FUNCTION_BLOCK FB_VALVE_X_3_PROP IMPLEMENTS I_VALVE_X_3_PROP
VAR_OUTPUT
  iAnalogSwitch:                                          INT;
END_VAR
VAR //General
	{attribute 'instance-path'} 
  {attribute 'noinit'} 
	strInstancePath:									                      STRING;
	bInit: 												                          BOOL:=TRUE;
	strFullObjectPath: 								                      STRING;
	stEvent:											                          ST_EVENT;
	bAck:												                            BOOL;
END_VAR
VAR   // From FB_init	
	itfLogEvents: 										                      I_HANDLE_EVENTS;
  itfOpMode:											                        I_OP_MODE;
END_VAR                                      				
VAR	// Step chain control                				
  eSeq, eLastSeq, eNextSeq:					                      E_SEQ_VALVE; 
                  				
  //eActiveSeqState, eLastActiveSeqState:                 E_SEQ_GENERAL;
	(*
  iInternalSeqStateCase, iLastInternalSeqStateCase:       INT:=0;       
	tonDelay, tonTimeOut, tonStepTime:						          TON;
	tDelay:													                        TIME := T#100MS;
	tTimeOut:												                        TIME := T#100MS;
	tTimeOutExt:											                      TIME := T#100MS;
	bDelayActive, bTimeOutActiveQuit, bTimeOutActiveNoQuit:	BOOL;//Timer Option
	bActiveStep, bDebugAcitve, bDebugNext:					        BOOL;//Debug Option
	i:														                          INT;
 	iError:													                        INT; //ERROR-CODE                    	                   		
	listLastSteps:											                    ARRAY[0..49] OF ST_LAST_STEPS;	
	strExtraInfo:											                      STRING; 
	eStep_Type:												                      E_STEP_STATE_TYPE; 
	bDebugModeActive:										                    BOOL;   
	bWaitForBreakpoint:										                  BOOL;
	bBreakpointActive:										                  BOOL;
	bDebugResume:											                      BOOL;   
	listBreakpoint:											                    ARRAY[0..10] OF  INT;    
*)
i:														                            INT;
stSeqCtrlGeneral:											                    ST_SEQ_CTRL_GEN;     	
END_VAR                                             		
VAR                                                 		
	bMethodeFromExtStarted:									                BOOL;
	bMethodeFromExtActive:									                BOOL;
	bMethodeFromExtDone:									                  BOOL;
	strTemp:												                        STRING;
END_VAR   
VAR
  stHMI:                                                  ST_HMI_VALVE;
  tDelay:                                                 TIME;
  rSpeedInPercent:                                        REAL;
END_VAR
VAR
  iOutputVal:                                             INT; 
END_VAR                 	
VAR_TEMP                    	
	iTemp:										                              INT;
END_VAR

// Set FBs and Interfaces ready after switch internal step
IF stSeqCtrlGeneral.iInternalSeqStateCase <> stSeqCtrlGeneral.iLastInternalSeqStateCase AND NOT stSeqCtrlGeneral.bExitSetReadyState THEN
  IF TRUE
  //AND ...
  THEN
    stSeqCtrlGeneral.bExitSetReadyState := TRUE;
  ELSE
    RETURN;
  END_IF
END_IF

stSeqCtrlGeneral.strObject := F_CreateObjectName(strInstancePath);

// First method call
_m_SequenceManager();
//_m_SaveLastStep();

CASE eSeq OF 
  E_SEQ_VALVE.BASE:;
  
	E_SEQ_VALVE.INIT: _m_Seq_INIT();
		IF TRUE
		AND (stSeqCtrlGeneral.eActiveSeqState = E_SEQ_GENERAL.DONE) 
		THEN
			eSeq := E_SEQ_VALVE.BASE;
		END_IF
		
	E_SEQ_VALVE.SETUP:;
  
	// Process
  E_SEQ_VALVE.SET_LIMIT: _m_Seq_VALVE_CTRL();
    IF TRUE
		AND (stSeqCtrlGeneral.eActiveSeqState = E_SEQ_GENERAL.DONE) 
		THEN
			eSeq := E_SEQ_VALVE.BASE;
		END_IF
    
  E_SEQ_VALVE.SET_LIMIT_SMOOTH: _m_Seq_VALVE_CTRL_SMOOTH();
    IF TRUE
		AND (stSeqCtrlGeneral.eActiveSeqState = E_SEQ_GENERAL.DONE) 
		THEN
			eSeq := E_SEQ_VALVE.BASE;
		END_IF

  // End
	E_SEQ_VALVE.END:;
	E_SEQ_VALVE.ERROR_SEQ:;	
END_CASE

strTemp:=TO_STRING(eSeq);

METHOD PRIVATE _m_DebugManager
VAR_INPUT
	iStepID: int;
END_VAR
IF TRUE
AND THIS^.stSeqCtrlGeneral.bDebugModeActive 
AND NOT THIS^.stSeqCtrlGeneral.bActiveStep
THEN


THIS^.stSeqCtrlGeneral.bBreakpointActive:=FALSE;

FOR i:=0 TO 10 DO
	
	IF TRUE
	AND iStepID=THIS^.stSeqCtrlGeneral.listBreakpoint[i] 
	AND iStepID<>0
	THEN
		EXIT;
	END_IF
END_FOR
IF (i<=10) THEN
	THIS^.stSeqCtrlGeneral.bBreakpointActive:=TRUE;
END_IF

END_IF
END_METHOD

METHOD PRIVATE _m_Delay : BOOL
VAR_INPUT
	DelayTime:	TIME;
END_VAR
THIS^.stSeqCtrlGeneral.bDelayActive:=TRUE;
THIS^.stSeqCtrlGeneral.tDelay:=DelayTime;
_m_Delay:=FALSE;
IF THIS^.stSeqCtrlGeneral.tonDelay.Q THEN
	_m_Delay:=TRUE;
END_IF
END_METHOD

METHOD PRIVATE _m_GeneralStepSetting : BOOL
VAR_INPUT
	StepType:			    	E_STEP_STATE_TYPE;
	InfoTextID:					STRING(20);
	EnableDebug:	   			BOOL;	
	
END_VAR
IF THIS^.stSeqCtrlGeneral.bActiveStep THEN
	THIS^.stSeqCtrlGeneral.eStep_Type:=StepType;
	THIS^.stSeqCtrlGeneral.strExtraInfo:= GenLib.F_RET_TXTLIST_ENTRY(strPortNr:='851',strID:='',strTxtLstName:=InfoTextID);
END_IF
END_METHOD

METHOD PRIVATE _m_SaveLastStep : BOOL
VAR_INPUT
END_VAR
VAR
	i: dint;
END_VAR
IF NOT THIS^.stSeqCtrlGeneral.bActiveStep THEN
	
	FOR i:=49 TO 1 BY -1 DO
			stSeqCtrlGeneral.listLastSteps[i].strStepName:=stSeqCtrlGeneral.listLastSteps[i-1].strStepName;
			stSeqCtrlGeneral.listLastSteps[i].tStepTime:=stSeqCtrlGeneral.listLastSteps[i-1].tStepTime;
			stSeqCtrlGeneral.listLastSteps[i].tDelayTime:=stSeqCtrlGeneral.listLastSteps[i-1].tDelayTime;
	END_FOR
	stSeqCtrlGeneral.listLastSteps[0].strStepName:=TO_STRING(THIS^.eSeq);
	stSeqCtrlGeneral.listLastSteps[1].tStepTime:=THIS^.stSeqCtrlGeneral.tonStepTime.ET;
	stSeqCtrlGeneral.listLastSteps[1].tStepTime:=THIS^.stSeqCtrlGeneral.tonDelay.ET;
ELSE
	stSeqCtrlGeneral.listLastSteps[0].tStepTime:=THIS^.stSeqCtrlGeneral.tonStepTime.ET;
	stSeqCtrlGeneral.listLastSteps[0].tDelayTime:=THIS^.stSeqCtrlGeneral.tonDelay.ET;	
END_IF
END_METHOD

METHOD PRIVATE _m_Seq_INIT : BOOL
VAR
  ActiveSeq: STRING;
END_VAR
//THIS^._m_GeneralStepSetting(StepType:=E_STEP_STATE_TYPE.INIT,
ActiveSeq := TO_STRING(THIS^.eSeq);

CASE THIS^.stSeqCtrlGeneral.eActiveSeqState OF
E_SEQ_GENERAL.READY:;

	
E_SEQ_GENERAL.EXECUTE:;
	IF TRUE
	THEN
		THIS^.stSeqCtrlGeneral.eActiveSeqState := E_SEQ_GENERAL.RESET;
	END_IF
  
E_SEQ_GENERAL.RESET:;
	stSeqCtrlGeneral.iInternalSeqStateCase := 0;
	IF TRUE
	THEN
		THIS^.stSeqCtrlGeneral.eActiveSeqState := E_SEQ_GENERAL.BUSY;
	END_IF
  
E_SEQ_GENERAL.BUSY:;
	CASE THIS^.stSeqCtrlGeneral.iInternalSeqStateCase OF
    0:  // Reset valve
      IF TRUE 
			THEN 
        iAnalogSwitch := 0;
        IF _m_Delay(T#1S) THEN
          THIS^.stSeqCtrlGeneral.iInternalSeqStateCase := 1000;
				END_IF
			END_IF
      
	ELSE
		THIS^.stSeqCtrlGeneral.eActiveSeqState := E_SEQ_GENERAL.DONE;  
	END_CASE
	THIS^.stSeqCtrlGeneral.strExtraInfo := CONCAT('Internal state: ', TO_STRING(THIS^.stSeqCtrlGeneral.iInternalSeqStateCase));

E_SEQ_GENERAL.DONE:;

E_SEQ_GENERAL.ERROR:;

E_SEQ_GENERAL.TIME_OUT:; 
IF TRUE
AND THIS^.stSeqCtrlGeneral.bTimeOutActiveQuit 
THEN
  THIS^.stSeqCtrlGeneral.strExtraInfo := 'Bitte quittieren und erneut testen';
  IF TRUE
  //AND itfOpMode.P_QUIT
  THEN
    THIS^.stSeqCtrlGeneral.eActiveSeqState := E_SEQ_GENERAL.EXECUTE;
	END_IF
  
END_IF

ELSE
  THIS^.stSeqCtrlGeneral.eActiveSeqState := E_SEQ_GENERAL.ERROR;
END_CASE
END_METHOD

METHOD PRIVATE _m_Seq_VALVE_CTRL : BOOL
VAR
  ActiveSeq:  STRING;
END_VAR
//THIS^._m_GeneralStepSetting(StepType:=E_STEP_STATE_TYPE.INIT,
ActiveSeq := TO_STRING(THIS^.eSeq);

CASE THIS^.stSeqCtrlGeneral.eActiveSeqState OF
E_SEQ_GENERAL.READY:;

	
E_SEQ_GENERAL.EXECUTE:;
	IF TRUE
	THEN
		THIS^.stSeqCtrlGeneral.eActiveSeqState := E_SEQ_GENERAL.RESET;
	END_IF
  
E_SEQ_GENERAL.RESET:;
	stSeqCtrlGeneral.iInternalSeqStateCase := 0;
	IF TRUE
	THEN
		THIS^.stSeqCtrlGeneral.eActiveSeqState := E_SEQ_GENERAL.BUSY;
	END_IF
  
E_SEQ_GENERAL.BUSY:;
	CASE THIS^.stSeqCtrlGeneral.iInternalSeqStateCase OF
    0:  // Calc output value
      IF TRUE 
			THEN 
        THIS^.iOutputVal := TO_INT(327.67 * THIS^.rSpeedInPercent);
        IF THIS^.iOutputVal < 0 THEN 
          THIS^.iOutputVal := THIS^.iOutputVal - 1;
        END_IF
        iAnalogSwitch := THIS^.iOutputVal;
        THIS^.stSeqCtrlGeneral.iInternalSeqStateCase := 10;
			END_IF
      
    10:  // Set output value
      IF TRUE 
			THEN 
        iAnalogSwitch := THIS^.iOutputVal;
        THIS^.stSeqCtrlGeneral.iInternalSeqStateCase := 1000;
			END_IF
      
	ELSE
		THIS^.stSeqCtrlGeneral.eActiveSeqState := E_SEQ_GENERAL.DONE;  
	END_CASE
	THIS^.stSeqCtrlGeneral.strExtraInfo := CONCAT('Internal state: ', TO_STRING(THIS^.stSeqCtrlGeneral.iInternalSeqStateCase));

E_SEQ_GENERAL.DONE:;

E_SEQ_GENERAL.ERROR:;

E_SEQ_GENERAL.TIME_OUT:; 
IF TRUE
AND THIS^.stSeqCtrlGeneral.bTimeOutActiveQuit 
THEN
  THIS^.stSeqCtrlGeneral.strExtraInfo := 'Bitte quittieren und erneut testen';
  IF TRUE
  //AND itfOpMode.P_QUIT
  THEN
    THIS^.stSeqCtrlGeneral.eActiveSeqState := E_SEQ_GENERAL.EXECUTE;
	END_IF
  
END_IF

ELSE
  THIS^.stSeqCtrlGeneral.eActiveSeqState := E_SEQ_GENERAL.ERROR;
END_CASE
END_METHOD

METHOD PRIVATE _m_Seq_VALVE_CTRL_SMOOTH : BOOL
VAR
  ActiveSeq:  STRING;
END_VAR
//THIS^._m_GeneralStepSetting(StepType:=E_STEP_STATE_TYPE.INIT,
ActiveSeq := TO_STRING(THIS^.eSeq);

CASE THIS^.stSeqCtrlGeneral.eActiveSeqState OF
E_SEQ_GENERAL.READY:;

	
E_SEQ_GENERAL.EXECUTE:;
	IF TRUE
	THEN
		THIS^.stSeqCtrlGeneral.eActiveSeqState := E_SEQ_GENERAL.RESET;
	END_IF
  
E_SEQ_GENERAL.RESET:;
	stSeqCtrlGeneral.iInternalSeqStateCase := 0;
	IF TRUE
	THEN
		THIS^.stSeqCtrlGeneral.eActiveSeqState := E_SEQ_GENERAL.BUSY;
	END_IF
  
E_SEQ_GENERAL.BUSY:;
	CASE THIS^.stSeqCtrlGeneral.iInternalSeqStateCase OF
    0:  // Calc output value
      IF TRUE 
			THEN 
        THIS^.iOutputVal := TO_INT(327.67 * THIS^.rSpeedInPercent);
        IF THIS^.iOutputVal < 0 THEN 
          THIS^.iOutputVal := THIS^.iOutputVal - 1;
        END_IF
        iAnalogSwitch := THIS^.iOutputVal;
        THIS^.stSeqCtrlGeneral.iInternalSeqStateCase := 10;
			END_IF
      
    10:  // Set output value
      IF TRUE 
			THEN 
        IF iAnalogSwitch > THIS^.iOutputVal + 100 THEN
          iAnalogSwitch := iAnalogSwitch - 100;
        ELSIF iAnalogSwitch < THIS^.iOutputVal - 100 THEN
          iAnalogSwitch := iAnalogSwitch + 100;
        END_IF
        IF ABS(iAnalogSwitch - THIS^.iOutputVal) <= 100 THEN
          THIS^.stSeqCtrlGeneral.iInternalSeqStateCase := 20;
        END_IF
			END_IF
      
    20:  // Set output value
      IF TRUE 
			THEN 
        iAnalogSwitch := THIS^.iOutputVal;
        THIS^.stSeqCtrlGeneral.iInternalSeqStateCase := 1000;
			END_IF
      
	ELSE
		THIS^.stSeqCtrlGeneral.eActiveSeqState := E_SEQ_GENERAL.DONE;  
	END_CASE
	THIS^.stSeqCtrlGeneral.strExtraInfo := CONCAT('Internal state: ', TO_STRING(THIS^.stSeqCtrlGeneral.iInternalSeqStateCase));

E_SEQ_GENERAL.DONE:;

E_SEQ_GENERAL.ERROR:;

E_SEQ_GENERAL.TIME_OUT:; 
IF TRUE
AND THIS^.stSeqCtrlGeneral.bTimeOutActiveQuit 
THEN
  THIS^.stSeqCtrlGeneral.strExtraInfo := 'Bitte quittieren und erneut testen';
  IF TRUE
  //AND itfOpMode.P_QUIT
  THEN
    THIS^.stSeqCtrlGeneral.eActiveSeqState := E_SEQ_GENERAL.EXECUTE;
	END_IF
  
END_IF

ELSE
  THIS^.stSeqCtrlGeneral.eActiveSeqState := E_SEQ_GENERAL.ERROR;
END_CASE
END_METHOD

METHOD PRIVATE _m_SequenceManager
VAR_INPUT
END_VAR
IF FALSE
//AND THIS^.eActiveSeqState=DONE 
AND eLastSeq<>eSeq
THEN
	IF THIS^.stSeqCtrlGeneral.eActiveSeqState<>E_SEQ_GENERAL.EXECUTE THEN
		THIS^.stSeqCtrlGeneral.eActiveSeqState:=E_SEQ_GENERAL.READY;
	END_IF
END_IF

eSeq := eNextSeq;

//DelayTimer und TimeOut Timer verwalten
stSeqCtrlGeneral.bActiveStep:=	TRUE
				AND eLastSeq					=	eSeq
				AND stSeqCtrlGeneral.eLastActiveSeqState			=	stSeqCtrlGeneral.eActiveSeqState
				AND	stSeqCtrlGeneral.iLastInternalSeqStateCase	=	stSeqCtrlGeneral.iInternalSeqStateCase
				;
			
IF NOT stSeqCtrlGeneral.bActiveStep THEN
	stSeqCtrlGeneral.bDelayActive:=FALSE;
	stSeqCtrlGeneral.bTimeOutActiveQuit:=FALSE;
	stSeqCtrlGeneral.bTimeOutActiveNoQuit:=FALSE;
  THIS^.stSeqCtrlGeneral.strExtraInfo:='';
END_IF

_m_SaveLastStep();
stSeqCtrlGeneral.tonDelay	(IN:=stSeqCtrlGeneral.bActiveStep AND stSeqCtrlGeneral.bDelayActive, 		PT:=stSeqCtrlGeneral.tDelay);
stSeqCtrlGeneral.tonTimeOut	(IN:=stSeqCtrlGeneral.bActiveStep AND (stSeqCtrlGeneral.bTimeOutActiveNoQuit OR stSeqCtrlGeneral.bTimeOutActiveQuit), 	PT:=stSeqCtrlGeneral.tTimeOut);
stSeqCtrlGeneral.tonStepTime	(IN:= stSeqCtrlGeneral.bActiveStep, PT:= T#24H);

IF stSeqCtrlGeneral.tonTimeOut.Q  THEN
	stSeqCtrlGeneral.eActiveSeqState:=E_SEQ_GENERAL.TIME_OUT;
END_IF

IF stSeqCtrlGeneral.iError<>0 THEN
	eSeq:=E_SEQ_VALVE.ERROR_SEQ;
END_IF



eLastSeq					:=	eSeq;
stSeqCtrlGeneral.eLastActiveSeqState			:=	stSeqCtrlGeneral.eActiveSeqState;
stSeqCtrlGeneral.iLastInternalSeqStateCase	:=	stSeqCtrlGeneral.iInternalSeqStateCase;

// Reset set ready state
IF THIS^.stSeqCtrlGeneral.bExitSetReadyState THEN
  THIS^.stSeqCtrlGeneral.bExitSetReadyState := FALSE;
END_IF
END_METHOD

METHOD PRIVATE _m_TimeOut : BOOL
VAR_INPUT
	bTimeoutActiveToQuit:	BOOL;
	bTimeOutActiveNoQuit:	BOOL;
	tTimeOut:				TIME;	
END_VAR
THIS^.stSeqCtrlGeneral.bTimeOutActiveQuit:=	bTimeoutActiveToQuit;
THIS^.stSeqCtrlGeneral.bTimeOutActiveNoQuit:=	bTimeOutActiveNoQuit;
THIS^.stSeqCtrlGeneral.tTimeOut:=			tTimeOut;
_m_TimeOut:=FALSE;
IF THIS^.stSeqCtrlGeneral.tonTimeOut.Q THEN
	_m_TimeOut:=TRUE;
END_IF
END_METHOD

METHOD FB_init : BOOL
VAR_INPUT
	bInitRetains : BOOL; // if TRUE, the retain variables are initialized (warm start / cold start)
	bInCopyCode : BOOL;  // if TRUE, the instance afterwards gets moved into the copy code (online change)
  
  itfLogEvents: 										                      I_HANDLE_EVENTS;
  itfOpMode:											                        I_OP_MODE; 
END_VAR
THIS^.itfLogEvents := itfLogEvents;
THIS^.itfOpMode := itfOpMode;
END_METHOD

METHOD M_Reset : BOOL
VAR_INPUT
END_VAR
M_Reset := THIS^.stSeqCtrlGeneral.eActiveSeqState = E_SEQ_GENERAL.DONE;

// Assign input

// General
IF THIS^.stSeqCtrlGeneral.eActiveSeqState = E_SEQ_GENERAL.READY THEN
  THIS^.eNextSeq := E_SEQ_VALVE.INIT;
  THIS^.stSeqCtrlGeneral.eActiveSeqState := E_SEQ_GENERAL.EXECUTE;
END_IF
END_METHOD

(*=== Method: M_Run  ============================================

 @brief: Here is the global code (Timer, Event, Flange,...)*)
METHOD M_Run
END_METHOD

METHOD M_SetReady : BOOL
VAR_INPUT
END_VAR
M_SetReady := TRUE
              AND THIS^.stSeqCtrlGeneral.eActiveSeqState = E_SEQ_GENERAL.READY
              AND THIS^.eSeq = E_SEQ_VALVE.BASE;

THIS^.stSeqCtrlGeneral.eActiveSeqState := E_SEQ_GENERAL.READY;
THIS^.eNextSeq := E_SEQ_VALVE.BASE;
END_METHOD

METHOD M_ValveCtrl : BOOL
VAR_INPUT
  /// -100 to -1 = Move to HP, 1 to 100 = Move to WP, 0 = Off
  rSpeedInPercent:        REAL;
  tDelay:                 TIME;
END_VAR
M_ValveCtrl := THIS^.stSeqCtrlGeneral.eActiveSeqState = E_SEQ_GENERAL.DONE;

// Assign input
IF rSpeedInPercent < -100 THEN
  rSpeedInPercent := -100;
ELSIF rSpeedInPercent > 100 THEN
  rSpeedInPercent := 100;
END_IF
THIS^.rSpeedInPercent := rSpeedInPercent;
THIS^.tDelay := tDelay;

// General
IF THIS^.stSeqCtrlGeneral.eActiveSeqState = E_SEQ_GENERAL.READY THEN
  THIS^.eNextSeq := E_SEQ_VALVE.SET_LIMIT;
  THIS^.stSeqCtrlGeneral.eActiveSeqState := E_SEQ_GENERAL.EXECUTE;
END_IF
END_METHOD

METHOD M_ValveCtrlSmooth : BOOL
VAR_INPUT
  /// -100 to -1 = Move to HP, 1 to 100 = Move to WP, 0 = Off
  rSpeedInPercent:        REAL;
  tDelay:                 TIME;
END_VAR
M_ValveCtrlSmooth := THIS^.stSeqCtrlGeneral.eActiveSeqState = E_SEQ_GENERAL.DONE;

// Assign input
IF rSpeedInPercent < -100 THEN
  rSpeedInPercent := -100;
ELSIF rSpeedInPercent > 100 THEN
  rSpeedInPercent := 100;
END_IF
THIS^.rSpeedInPercent := rSpeedInPercent;
THIS^.tDelay := tDelay;

// General
IF THIS^.stSeqCtrlGeneral.eActiveSeqState = E_SEQ_GENERAL.READY THEN
  THIS^.eNextSeq := E_SEQ_VALVE.SET_LIMIT_SMOOTH;
  THIS^.stSeqCtrlGeneral.eActiveSeqState := E_SEQ_GENERAL.EXECUTE;
END_IF
END_METHOD

{warning 'Eigenschaftenimplementierung hinzufügen'}
PROPERTY P_CurrentVal : INT
GET
P_CurrentVal := THIS^.iOutputVal;
END_GET
END_PROPERTY

(*=== Property: P_Event  ============================================

 @param [set]: 	Set the Structure "ST_EVENT" from another Object
 @param [get]: 	Return the Structure "ST_EVENT", it contains the actual 
					event of the Object *)
PROPERTY P_Event : GenLib.ST_EVENT
GET
END_GET
SET
END_SET
END_PROPERTY

{warning 'Eigenschaftenimplementierung hinzufügen'}
(*=== Property: P_FullObjectPath  ============================================

 @param [set]: 	Set the Object Path (Clear String of Object)
 @param [get]: 	Return the Objectpath *)
PROPERTY P_FullObjectPath : STRING
GET
END_GET
SET
END_SET
END_PROPERTY

{warning 'Eigenschaftenimplementierung hinzufügen'}
(*=== Property: P_Global_Ack  ============================================

 @param [set]: 	Set the Bit for Ack from another Object
 @param [get]: 	Return the state of Ack Bit*)
PROPERTY P_Global_Ack : BOOL
GET
END_GET
SET
END_SET
END_PROPERTY

{warning 'Eigenschaftenimplementierung hinzufügen'}
(*=== Property: P_GlobalID  ============================================

 @param [set]: 	-
 @param [get]: 	Return the string of instance path*)
PROPERTY P_GlobalID : STRING
GET
END_GET
END_PROPERTY

{warning 'Eigenschaftenimplementierung hinzufügen'}
PROPERTY P_ReadyState : BOOL
GET
P_ReadyState := THIS^.stSeqCtrlGeneral.eActiveSeqState = E_SEQ_GENERAL.READY;
END_GET
END_PROPERTY

PROPERTY P_SpeedInPercent : REAL
GET
P_SpeedInPercent := THIS^.rSpeedInPercent;
END_GET
END_PROPERTY

END_FUNCTION_BLOCK

(* stored: Version 1.1.0.1, ProductVersion 3.1.4024.12
   POU FB_VALVE_X_3_PROP: Id {482439bb-28b1-4541-8ef1-944c797b650d}, SpecialFunc None
   Folder PRIVAT: Id {05d28711-59e2-48db-8558-5a7de7e344de}
   Folder SEQUENCE: Id {31d0de76-8fa9-474c-baaf-3618880ee38e}
   Method _m_DebugManager: Id {0b60cd08-e6dc-49dd-8482-7d957c76693a}
   Method _m_Delay: Id {43c81bee-e6f7-4c5d-8b1f-997ad3fbc35e}
   Method _m_GeneralStepSetting: Id {a128ee0c-20b1-4f69-a3df-6e9a05d23cfa}
   Method _m_SaveLastStep: Id {eae4279d-d981-40a1-8696-108e337fbb2c}
   Method _m_Seq_INIT: Id {cf7a0ba0-1554-45bc-b419-e35652801c01}
   Method _m_Seq_VALVE_CTRL: Id {6b6f5e0c-6701-4e55-9491-20e3af6803d5}
   Method _m_Seq_VALVE_CTRL_SMOOTH: Id {82ab1a1e-1052-412b-baa0-ce2414221aa9}
   Method _m_SequenceManager: Id {4a0583b9-78d0-43d5-b811-9e03a84aab50}
   Method _m_TimeOut: Id {43abcb32-0942-46b6-9874-a24d7a2d241e}
   Method FB_init: Id {bc03c7f8-6622-4106-a379-11ee8752b89a}
   Method M_Reset: Id {a8c3f74a-28b6-4c1f-a3ff-52aafc54b192}
   Method M_Run: Id {1b360013-34ab-4a10-bcdd-060fe0b772be}
   Method M_SetReady: Id {12f7a4c6-269a-49ae-8b49-49973a7973b4}
   Method M_ValveCtrl: Id {76f55699-99d6-4d52-8a45-744a3b70ad2f}
   Method M_ValveCtrlSmooth: Id {ef3691b5-0cf8-4a4e-9723-664fe51cd119}
   Property P_CurrentVal: Id {b1db8223-9bf9-45db-afa5-673a7131351b}
   Get Get: Id {5422843c-bc6b-4a2f-89d9-bfa6f97cba06}
   Property P_Event: Id {af008fdf-e329-49af-9931-f0d5ed8a0f21}
   Get Get: Id {d47b9bae-4e00-4930-93ed-cb6db512b602}
   Set Set: Id {92b27336-2b2f-4f1f-b81a-bc5cdbe376ff}
   Property P_FullObjectPath: Id {a2e2efe2-acd5-4883-afd2-732293ea362c}
   Get Get: Id {0ef6ed5c-8d09-4f90-a9d8-eebefebb8ea6}
   Set Set: Id {28c46471-21e0-4fea-b301-ff81d48ae610}
   Property P_Global_Ack: Id {7654c778-d6f0-4d5f-aca5-324c22d6c51c}
   Get Get: Id {0cb4bd8a-4b21-440d-a882-f1e29d214e46}
   Set Set: Id {2cc25148-464c-4113-a557-c0b99a780470}
   Property P_GlobalID: Id {71d1c867-c580-4fd8-8083-861dc06f0b4d}
   Get Get: Id {41d05e68-57a4-404b-9543-8d2f89f9e1ad}
   Property P_ReadyState: Id {59f97911-63ed-446e-a1d0-f2962d43dd64}
   Get Get: Id {af481d79-9e87-4799-89ee-11fb13cf8f67}
   Property P_SpeedInPercent: Id {6d3e229a-4c7d-4baa-8879-f01351c40716}
   Get Get: Id {e020cdc9-e10e-4fb8-b04a-12c7c81fdfa9} *)
